PROGRAM PRG_ST1K1_ZOS
VAR
END_VAR

END_PROGRAM

(* stored: Version 1.1.0.1, ProductVersion 3.1.4022.18
   POU PRG_ST1K1_ZOS: Id {ddf40798-9a4a-4d46-9d44-fa3eb642a3fd}, SpecialFunc None *)
